TYPE ST_TransportDataEmulation :
(**************************************************************************************
 * 	Application		:	BoxControl Framework
 *	Revision		:	$Revision: 404529 $
 *	Revision date	:	$Date: 2018-04-23 08:21:38 +0200 (Mo., 23 Apr 2018) $
 *	Last changed by	:	$Author: b7bolm $
 *	URL				:	$URL: http://almscdc.swisslog.com/repo/SWPD/Development/BoxControlFramework/20_Release/trunk/01_Software/BCF/BCF/JumpStart/20_Product/11_Emu/12_E_Functions/10_Lib/10_Conv/01_DUTs/ST_TransportDataEmulation.TcDUT $
 *
 *	Purpose			:	Transport control data
 *
 * ------------------------------------------------------------------------------------
 *	Copyright Swisslog [IP AG], Switzerland. All rights reserved.
 * 
 * ------------------------------------------------------------------------------------
 *	
 * 	Revision History: 
 *
 * 	VERSION			DATE			INITIALS			DESCRIPTION
 *	0.1				01.01.2001		swl					Example
 *
 **************************************************************************************)	
STRUCT
	eFunctionNumber			: E_FunctionNumber; // Number oft the function
	ZoneNumber 				: INT;
	rSettings 				: REFERENCE TO ST_CFG_Zone;
	rTransportControlData	: REFERENCE TO ST_TransportControlDataEmulation;
	rRealObjTrspControlData	: REFERENCE TO ST_TransportControlData;
END_STRUCT
END_TYPE

(* stored: Version 1.1.0.1, ProductVersion 3.1.4022.12
   DUT ST_TransportDataEmulation: Id {fc80a3a5-7a11-4fa5-96a6-c5efd0d22831} *)
